TYPE AnyType : __SYSTEM.TYPE_CLASS; END_TYPE

(* stored: Version 1.1.0.1
   DUT AnyType: Id {172f50c8-14c6-0d20-0444-a6b912ac2017} *)
